FUNCTION_BLOCK T_MockNumberCommandTask IMPLEMENTS I_NumberResultTask
VAR_INPUT
  _Busy, _Done, _Error, _Timeout : BOOL;
  _Result : LREAL;
END_VAR

METHOD Abort
END_METHOD

PROPERTY Available : BOOL
GET
END_GET
END_PROPERTY

PROPERTY Busy : BOOL
GET
Busy := _Busy;
END_GET
END_PROPERTY

METHOD CyclicLogic
END_METHOD

PROPERTY Done : BOOL
GET
Done := _Done;
END_GET
END_PROPERTY

PROPERTY Error : BOOL
GET
Error := _Error;
END_GET
END_PROPERTY

PROPERTY ErrorId : STRING
GET
END_GET
END_PROPERTY

METHOD Execute : BOOL
END_METHOD

METHOD Free
END_METHOD

PROPERTY Result : LREAL
GET
Result := _Result;
END_GET
END_PROPERTY

PROPERTY Timeout : BOOL
GET
Timeout := _Timeout;
END_GET
END_PROPERTY

END_FUNCTION_BLOCK

(* stored: Version 1.1.0.1
   POU T_MockNumberCommandTask: Id {c4b4e451-f370-4703-94b5-7d62d9b1c95d}, SpecialFunc None
   Method Abort: Id {c650fcad-4301-4238-b126-680f55041cbb}
   Property Available: Id {56da4a8e-a5ae-4aab-ae87-ec2b15a18fc6}
   Get Get: Id {7df23a0e-c48f-49ac-ae9f-b3593db904c8}
   Property Busy: Id {72c90843-3c63-4da2-9393-dcb91570b44e}
   Get Get: Id {d9b4099c-f991-4541-825e-b7957299caa3}
   Method CyclicLogic: Id {fa2ae519-8201-44d1-8710-f9947170a4d0}
   Property Done: Id {030e85d9-0e29-47d2-8ccf-d322f4e300f1}
   Get Get: Id {736d6366-48e0-4555-abc9-a51a5699281f}
   Property Error: Id {48d37403-a39e-4a16-8663-73c985b8a52b}
   Get Get: Id {5bffc08d-d734-4d55-8ec5-e1702df6fbec}
   Property ErrorId: Id {3e0e85d2-fbf4-4dce-8d66-ea33175aa12c}
   Get Get: Id {1de7f265-5462-4327-bbd3-e76ce62be1bf}
   Method Execute: Id {515bc31e-479f-4fb8-9310-a221689dccc1}
   Method Free: Id {4765e9db-1340-4adf-aab2-4785b6036cb8}
   Property Result: Id {4f59f975-8b8b-4e6f-9705-8fba422beb9c}
   Get Get: Id {5f2cfd92-2a40-4d37-82a2-83afcc6cf8dc}
   Property Timeout: Id {a0367408-d28c-4fc7-a493-ff5cc1bbce82}
   Get Get: Id {71bd9546-6b81-4425-869e-2ea66e778e37} *)
